// SIMATIC S7-200 project (STEP 7-Micro/WIN), CPU 226 REL 01.22

SYMBOL_TABLE USR1
Always_On        SM0.0    // This bit is always on.
First_Scan_On    SM0.1    // This bit is on for the first scan cycle only.
Clock_1s         SM0.5    // Clock pulse that is on for 0.5 s, off for 0.5 s, for a duty cycle time of 1 s.
Pot0_Value       SMB28    // Stores value entered by analog adjustment 0. Updated once per cycle in STOP/RUN
END_SYMBOL_TABLE

ORGANIZATION_BLOCK MAIN:OB1
TITLE=The system initializes on first startup, setting the TD 200 display state to 0 to show date and time, while initializing the pressure update speed to 50 (500ms), the pressure value to 12,345,678, and the output configuration to 0. Operators can use the TD 200 arrow keys to switch the display state, viewing different information such as date/time, pressure value, or motor status, with the state cycling between 0 and 6.
// When the display state is 1, operators can control pressure value updates via function keys F1-F4: F1 stops updates, F2 starts updates, F3 sets the update speed to 1 (10ms), and F4 sets it to 150 (1500ms). Pressure value updates are managed by a control flag and increment when the timer expires.
// If the display state is 2, F1 clears the output configuration to disable output points, F2 sets it to fully enabled, and F3 activates I/O cycling. The output configuration is set to fully enabled on the clock pulse rising edge and cleared on the falling edge.
// When the display state is 3, the system displays the analog potentiometer value in bar graph and numeric formats. For display state 4, the system supports scrolling message display, with F1-F4 setting the scroll speed to 1 (100ms), 5 (500ms), 10 (1000ms), or 15 (1500ms). In display state 6, it shows "ON 1" or "OFF 0" based on the motor status.
// The system supports a second TD 200 panel, with its display state controlling the content. State 0 shows the input byte in hexadecimal, decimal, and individual bit status, while state 1 shows the output byte’s equivalent information. 
BEGIN
Network 1 //  Initialize the Values to Be Used
//  Load SM0.1 to process this network in the first scan cycle only.
//  Move the hexadecimal value 8000 (binary 1000 0000 0000 0000) to variable
//  memory word VW12 to enable the first message on the TD 200 (device 1).
//  Move the constant 0 to variable memory word VW700 to set the
//  display state of the TD 200 to evaluate the function keys for
//  the pressure value (executed in subroutine SBR1).
//  Move the constant 0 to memory byte MB0 to clear the TD 200 function
//  key area.
//  Move the constant 0 to memory byte MB1 to clear the TD 200 help bit area.
//  Move the constant 50 to variable memory word VW704 to initialize
//  the embedded value for the pressure update speed.
//  Move the constant 12,345,678 to variable memory double word VD156
//  to set the pressure value.
//  Move the constant 0 to variable memory word VW706 to initialize
//  the output configuration with the function keys.
//  Fill the message area with full blocks in a bar graph.
//  Move 20 bytes starting from variable memory byte VB260 into VB900 to
//  copy the message to scroll on the TD 200 display.
//  Move the constant 15 to variable memory word VW800 to set the update
//  speed for the message scroll to slow.
//  Move the real number 1234.000 to variable memory double word VD316
//  to initialize the real value.
//  Move the hexadecimal value 80 (binary 1000 0000) to variable memory
//  byte VB512 to enable the second TD 200 (optional).
//  Move the constant 0 to variable memory word VW702 to set the
//  display state of the second TD 200 to zero.
// 
LD     First_Scan_On:SM0.1   // In the first scan cycle,
MOVW   16#8000, VW12         // enable the first message on
// device 1.
MOVW   +0, VW700             // Display the state of device 1
// set to zero.
MOVB   16#0, MB0             // Clear the function key area.
MOVB   16#0, MB1             // Clear the help bit area.
MOVW   +50, VW704            // Initialize the update speed (pressure)
MOVD   +12345678, VD156      // Set the pressure value.
MOVW   +0, VW706             // Initialize the I/O cycles.
FILL   16#FFFF, VW770, 10    // Fill the TD 200 message area
// with full blocks.
BMB    VB260, VB900, 20      // Copy the message to scroll.
MOVW   +15, VW800            // Set the scrolling update speed
// to slow.
MOVR   1234.0, VD316         // Initialize the real value.
MOVB   16#80, VB512          // Enable the first message on device
// 2.
MOVW   +0, VW702             // Set the display state of device
// 2 to zero.
Network 2 //  Set Up a Timer to Increment the Data Values
//  Load memory bit M1.0 to process this network (run the timer) only
//  when the pressure updates are running.
//  Start the retentive on-delay timer T1 with a preset time of the
//  value in variable memory word VW704. T1 has a resolution of 10 ms.
//  Each count of the current value is a multiple of that resolution.
//  For example, a count of 50 on a 10 ms timer represents 500 ms.
// 
LD     M1.0                  // Run timer only when the pressure
// updates are running.
TONR   T1, VW704             // Start timer T1 with a preset
// time of the value in VW704.
Network 3 //  Reset Timer T1 and Increment the Pressure Value
//  Load retentive on-delay timer T1 to process this network if the
//  timer has expired.
//  If the timer has expired,
//  reset the timer and
//  increment variable memory double word VD156 to increment the pressure
//  value.
// 
LD     T1                    // If timer T1 has expired,
R      T1, 1                 // reset the timer and
INCD   VD156                 // increment the pressure value.
Network 4 //  Subroutine SBR7
//  Special memory bit SM0.5 provides a clock pulse that is on for
//  0.5 s and off for 0.5 s, for a duty cycle time of 1 s.
//  Load SM0.5.
//  If there is a positive transition (Edge Up) at SM0.5,
//  move the hexadecimal value FFFF (binary 1111 1111 1111 1111) to variable
//  memory word VW706 to fill VW706 with ones and turn on the associated
//  outputs.
//  This subroutine writes a different text to the display, depending
//  on the status of input bit I0.0 (display state 6).
//  Start SBR6.
//  This subroutine reads the CPU input byte IB0 and displays
//  it in decimal format. The subroutine also displays the status of
//  each input bit (ON = 1, OFF = 0) on the TD 200 (device 2 display
//  state 0).
//  Start SBR7.
// 
LD     Clock_1s:SM0.5        // If the 0.5 s clock pulse value
EU                           // changes from 0 to 1,
MOVW   16#FFFF, VW706        // fill VW706 with ones to cycle
// on the outputs.
Network 5 //  Subroutine SBR4
//  Load SM0.5.
//  If there is a negative transition (Edge Down) at SM0.5,
//  move the hexadecimal value 0 to variable memory word VW706 to fill
//  VW706 with zeros and turn off the associated outputs.
//  This subroutine handles the memory bits set by the
//  TD 200 function keys (display state 1).
//  Start SBR1.
//  This subroutine writes a text message on the first row of the
//  TD 200 display and scrolls it to the left at the speed selected
//  (display state 4).
//  Start SBR4.
// 
LD     Clock_1s:SM0.5        // If the 0.5 s clock pulse value
ED                           // changes from 1 to 0,
MOVW   16#0, VW706           // fill VW706 with zeros to cycle
// off the outputs.
Network 6 //  Write the Values in Variable Memory Word VW706 to Outputs
//  Load memory bit M1.2 to process this network if the I/O cycle
//  process is enabled.
//  Move the value in VW706 to output word QW0.
// 
LD     M1.2                  // If the I/O cycles are enabled,
MOVW   VW706, QW0            // write to the outputs.
Network 7 //  If the TD 200 Display State Is 0, Call Subroutine SBR0
//  If the value in variable memory word VW700 is 0 (TD 200 menu 1 selected),
//  call subroutine SBR0 to display the date and time.
// 
LDW=   VW700, +0             // If the TD 200 display state = 0,
CALL   SBR_0:SBR0            // call SBR0.
Network 8 //  Subroutine SBR3
//  Check the value in memory byte MB0 to see if a function key on the
//  TD 200 has been pressed.
//  If the value in memory byte MB0 is not equal to 0
//  and the value in variable memory word VW700 is 1 (TD 200 menu 2 selected),
//  call subroutine SBR1 to evaluate the function keys to change
//  the pressure value.
//  This subroutine handles the function keys for the output configuration
//  (display state 2).
//  Start SBR2.
//  This subroutine contains the logic to display the analog adjustment
//  (POT) 0 in the form of a bar chart (display state 3). You can use
//  a small screwdriver to change the value of the POT.
//  Start SBR3.
// 
LDB=   MB0, 0                // If a function key
NOT                          // is pressed (MB0 not equal 0)
AW=    VW700, +1             // and the TD 200 display state  = 1,
CALL   SBR_1:SBR1            // call SBR1.
Network 9 //  If the TD 200 Display State Is 2, Call Subroutine SBR2
//  Check the value in memory byte MB0 to see if a function key on the
//  TD 200 has been pressed.
//  If the value in memory byte MB0 is not equal to 0
//  and the value in variable memory word VW700 is 2 (TD 200 menu 3 selected),
//  call subroutine SBR2 to evaluate the function keys to for the
//  output configuration.
// 
LDB=   MB0, 0                // If a function key
NOT                          // is pressed (MB0 not equal 0)
AW=    VW700, +2             // and the TD 200 display state = 2,
CALL   SBR_2:SBR2            // call SBR2.
Network 10 //  Subroutine SBR5
//  If the value in variable memory word VW700 is 3 (TD 200 menu 4 selected),
//  call subroutine SBR3 to update the analog adjustment (POT) value
//  as a bar chart graphic and in decimal form.
//  This subroutine clears the memory bits associated with the
//  TD 200 function keys. This allows a TD 200 system routine to edit
//  a real value after the ENTER key is pressed (display state 5).
//  Start SBR5.
// 
LDW=   VW700, +3             // If the TD 200 display state = 3,
CALL   SBR_3:SBR3            // call SBR3.
Network 11 //  If the TD 200 Display State Is 4, Call Subroutine SBR4
//  If the value in variable memory word VW700 is 4 (TD 200 menu 5 selected),
//  call subroutine SBR4 to scroll and display a message on the TD 200.
// 
LDW=   VW700, +4             // If the TD 200 display state = 4,
CALL   SBR_4:SBR4            // call SBR4.
Network 12 //  If the TD 200 Display State Is 5, Call Subroutine SBR5
//  If the value in variable memory word VW700 is 5 (TD 200 menu 6 selected),
//  call subroutine SBR5 to clear the memory bits of the function
//  keys.
// 
LDW=   VW700, +5             // If the TD 200 display state = 5,
CALL   SBR_5:SBR5            // call SBR5.
Network 13 //  Subroutine SBR8
//  If the value in variable memory word VW700 is 6 (TD 200 menu 7 selected),
//  call subroutine SBR6 to display the state of the motor (ON/OFF) on
//  the TD 200.
//  This subroutine reads the CPU output byte QB0 and displays
//  it in decimal format. The subroutine also displays the status of
//  each output bit (ON = 1, OFF = 0) on the TD 200 (device 2 display
//  state 1).
//  Start SBR8.
// 
LDW=   VW700, +6             // If the TD 200 display state = 6,
CALL   SBR_6:SBR6            // call SBR6.
Network 14 //  If the Second TD 200 Display State Is 0, Call Subroutine SBR7
//  If the value in variable memory word VW702 is 0 (second TD 200 menu
//  1 selected),
//  call subroutine SBR7 to update and display the CPU inputs.
// 
LDW=   VW702, +0             // If the second TD 200 display
// state = 0,
CALL   SBR_7:SBR7            // call SBR7.
Network 15 //  If the Second TD 200 Display State Is 1, Call Subroutine SBR8
//  If the value in variable memory word VW702 is 1 (second TD 200
//  menu 2 selected),
//  call subroutine SBR8 to update and display the CPU outputs.
// 
LDW=   VW702, +1             // If the second TD 200 display
// state = 1,
CALL   SBR_8:SBR8            // call SBR8.
Network 16 //  If the UP ARROW Is Pressed, Increment the Display State
//  Evaluate the arrow keys of the TD 200 device 1.
//  The first parameter block begins at VW0. The arrow keys are associated
//  with the fourth byte of the parameter block.
//  Load variable memory bit V3.3 to evaluate the UP ARROW key of the
//  TD 200.
//  If the UP ARROW key is pressed,
//  reset variable memory bit V3.3 and
//  increment variable memory word VW700 to change to the next TD 200
//  display state (move to the next TD 200 menu)
// 
LD     V3.3                  // If the UP ARROW key is pressed,
R      V3.3, 1               // reset V3.3 and
INCW   VW700                 // increment VW700.
Network 17 //  If the TD 200 Display State Moves above 6, Reset to 0
//  If the display state of the TD 200 = 7,
//  move the constant 0 to variable memory bit VW700 to change the
//  display state to 0.
// 
LDW=   VW700, +7             // If VW700 = 7,
MOVW   +0, VW700             // set the TD 200 display state = 0.
Network 18 //  If the DOWN ARROW Is Pressed, Decrement the Display State
//  Evaluate the arrow keys of the TD 200 device 1.
//  The first parameter block begins at VW0, The arrow keys are associated
//  with the fourth byte of the parameter block.
//  Load variable memory bit V3.2 to evaluate the DOWN ARROW key of the
//  TD 200.
//  If the DOWN ARROW key is pressed,
//  reset variable memory bit V3.2 and
//  decrement variable memory word VW700 to change to the previous TD 200
//  display state (move to the previous TD 200 menu)
// 
LD     V3.2                  // If the DOWN ARROW key is pressed,
R      V3.2, 1               // reset V3.2 and
DECW   VW700                 // decrement VW700.
Network 19 //  If the TD 200 Display State Moves below 0, Reset to 6
//  If the display state of the TD 200 = -1,
//  move the constant 6 to VW700 to change the display state to 6.
// 
LDW<=  VW700, -1             // If VW700 = -1,
MOVW   +6, VW700             // set the TD 200 display state = 6.
Network 20 //  If the UP ARROW Is Pressed, Increment the Display State of the Second Device
//  Evaluate the arrow keys of the TD 200 device 2.
//  The second device parameter block begins at VW500, The arrow
//  keys are associated with the fourth byte of the parameter block.
//  Load variable memory bit V503.3 to evaluate the UP ARROW key of the
//  second TD 200.
//  If the UP ARROW key is pressed,
//  reset variable memory bit V503.3 and
//  increment variable memory word VW702 to change to the next TD 200
//  display state (move to the next TD 200 menu)
// 
LD     V503.3                // If the UP ARROW key is pressed,
R      V503.3, 1             // reset V503.3 and
INCW   VW702                 // increment VW702.
Network 21 //  If the Second TD 200 Display State Moves above 1, Reset to 0
//  If the display state of the second TD 200 = 2,
//  move the constant 0 to variable memory bit VW702 to change the
//  display state to 0.
// 
LDW=   VW702, +2             // If VW702 = 2,
MOVW   +0, VW702             // set the TD 200 display state = 0.
Network 22 //  If the DOWN ARROW Is Pressed, Decrement the Display State of the Second Device
//  Evaluate the arrow keys of the TD 200 device 2.
//  The first parameter block begins at VW500, The arrow keys are associated
//  with the fourth byte of the parameter block.
//  Load variable memory bit V503.2 to evaluate the DOWN ARROW key of the
//  TD 200.
//  If the DOWN ARROW key is pressed,
//  reset variable memory bit V503.2 and
//  decrement variable memory word VW702 to change to the previous TD 200
//  display state (move to the previous TD 200 menu).
// 
LD     V503.2                // If the DOWN ARROW key is pressed,
R      V503.2, 1             // reset V503.2 and
DECW   VW702                 // decrement VW702.
Network 23 //  If the TD 200 Display State Moves below 0, Reset to 1
//  If the display state of the second TD 200 = -1,
//  move the constant 1 to VW702 to change the display state to 1.
// 
LDW<=  VW702, -1             // If VW702 = -1,
MOVW   +1, VW702             // set the TD 200 diplay state = 1.
Network 24 //  Set the Message Enable Bit Based on the Current Display State
//  Load special memory bit SM0.0 to process this network every scan cycle.
//  Move the hexadecimal value 8000 (binary 1000 0000 0000 0000) to
//  variable memory word VW12 to set the first message enable bit (V12.7)
//  Shift the value in VW12 by the value in variable memory byte VB701
//  (least significant byte of the display state variable memory word).
//  This sets the message enable bit that corresponds to the display state.
// 
LD     Always_On:SM0.0       // Every scan cycle,
MOVW   16#8000, VW12         // enable the first message
// on device 1.
SRW    VW12, VB701           // Shift the value in VW12 based on
// the value in VB701.
Network 25 //  Set the Message Enable Bit Based on the Current Display State of Device 2
//  Load special memory bit SM0.0 to process this network every scan cycle
//  Move the hexadecimal value 8000 (binary 1000 0000 0000 0000) to
//  variable memory word VW512 to set the first message enable bit (V512.7)
//  for the second TD 200 device.
//  Shift the value in VW512 by the value in variable memory byte VB703
//  (lest significant byte of the display state variable memory word).
//  This sets the message enable bit that corresponds to the display state
//  of the second device.
// 
LD     Always_On:SM0.0       // Every scan cycle,
MOVW   16#8000, VW512        // enable the first message
// on device 2.
SRW    VW512, VB703          // Shift the value in VW512 based on
// the value in VB703.
Network 26 //  Main Program End
//  End the main program.
// MEND					// End the main program.
// 
// ***SUBROUTINES***
// 
// 
Network 27 //  Subroutine SBR0
//  Start SBR0 to display the date and time on the TD 200 device 1.
// 
END_ORGANIZATION_BLOCK

SUBROUTINE_BLOCK SBR_0:SBR0
TITLE=
BEGIN
Network 2 //  Get and Display the Date
//  Load special memory bit SM0.0 to process this network every scan cycle.
//  Read the current time and date and load it in variable memory
//  byte VB720.
//  Starting at variable memory byte VB721, convert two hexadecimal digits
//  to an ASCII string and store the result at variable memory byte
//  VB100. This converts the month for display on the TD 200.
//  Move the hexadecimal value 2D to variable memory byte VB102 to
//  load a "-" to the TD 200 display.
//  Starting at variable memory byte VB722, convert two hexadecimal digits
//  to an ASCII string and store the result at variable memory byte
//  VB103. This converts the day of the month for display on the TD 200.
//  Move the hexadecimal value 2D to variable memory byte VB105 to
//  load a "-" to the TD 200 display.
//  Starting at variable memory byte VB720, convert two hexadecimal digits
//  to an ASCII string and store the result at variable memory byte
//  VB106. This converts the year for display on the TD 200.
//  Move the hexadecimal value 2020 to variable memory word VW108 to
//  load two blank spaces to the TD 200 display.
//  Move the hexadecimal value 2020 to variable memory word VW110 to
//  load two more blank spaces to the TD 200 display.
// 
LD     Always_On:SM0.0       // Every scan cycle,
TODR   VB720                 // read the real-time clock.
HTA    VB721, VB100, 2       // Convert the month to ASCII
// and display on the TD 200.
MOVB   16#2D, VB102          // Load a "-" for display.
HTA    VB722, VB103, 2       // Convert the day of the month
// and display.
MOVB   16#2D, VB105          // Load a "-" for display.
HTA    VB720, VB106, 2       // Convert the year to ASCII
// and display.
MOVW   16#2020, VW108        // Load two blanks.
MOVW   16#2020, VW110        // Load two blanks.
Network 3 //  Get and Display the Time
//  Load special memory bit SM0.0 to process this network every scan cycle.
//  Starting at variable memory byte VB723, convert two hexadecimal digits
//  to an ASCII string and store the result at variable memory byte
//  VB112. This converts the hour for display on the TD 200.
//  Move the hexadecimal value 3A to variable memory byte VB114 to
//  load a ":" to the TD 200 display.
//  Starting at variable memory byte VB724, convert two hexadecimal digits
//  to an ASCII string and store the result at variable memory byte
//  VB115. This converts the minutes for display on the TD 200.
//  Move the hexadecimal value 3A to variable memory byte VB117 to
//  load a ":" to the TD 200 display.
//  Starting at variable memory byte VB725, convert two hexadecimal digits
//  to an ASCII string and store the result at variable memory byte
//  VB118. This converts the seconds for display on the TD 200.
// 
LD     Always_On:SM0.0       // Every scan cycle,
HTA    VB723, VB112, 2       // convert the hour to ASCII
// and display on the TD 200.
MOVB   16#3A, VB114          // Load a ":" for display.
HTA    VB724, VB115, 2       // Convert the minutes to ASCII
// and display on the TD 200.
MOVB   16#3A, VB117          // Load a ":" for display.
HTA    VB725, VB118, 2       // Convert the seconds to ASCII
// and display on the TD 200.
Network 4 //  End of Subroutine SBR0
//  End SBR0.
// RET					// End SBR0.
// 
END_SUBROUTINE_BLOCK

SUBROUTINE_BLOCK SBR_1:SBR1
TITLE=
BEGIN
Network 2 //  Press F1 to Stop the Pressure Updates
//  Load memory bit M0.0 to check the status of the TD 200 function
//  key F1.
//  If memory bit M0.0 is set (F1 function key was pressed),
//  reset memory bit M1.0 to stop the pressure updates.
// 
LD     M0.0                  // If the F1 key has been pressed,
R      M1.0, 1               // stop the pressure updates.
Network 3 //  Press F2 to Start the Pressure Updates
//  Load memory bit M0.1 to check the status of the TD 200 function
//  key F2.
//  If memory bit M0.1 is set (F2 function key was pressed),
//  set memory bit M1.0 to start the pressure updates.
// 
LD     M0.1                  // If the F2 key has been pressed,
S      M1.0, 1               // start the pressure updates.
Network 4 //  Press F3 to Set the Pressure Readings for Fast Updates
//  Load memory bit M0.2 to check the status of the TD 200 function
//  key F3.
//  If memory bit M0.2 is set (F3 function key was pressed),
//  move the constant 1 to variable memory word VW704 to set the pressure
//  update speed to fast.
//  The value in VW704 is used as the preset time in the retentive
//  on-delay timer T1 (see Network 2). T1 has a resolution of 10 ms.
//  This means that a preset time (PT) of 1 results in a 10-ms timer.
// 
LD     M0.2                  // If the F3 key has been pressed,
MOVW   +1, VW704             // set the pressure readings for
// fast updates (10 ms).
Network 5 //  Press F4 to Set the Pressure Readings for Slow Updates
//  Load memory bit M0.3 to check the status of the TD 200 function
//  key F4.
//  If memory bit M0.3 is set (F4 function key was pressed),
//  move the constant 150 to variable memory word VW704 to set the pressure
//  update speed to slow.
//  The value in VW704 is used as the preset time in the retentive
//  on-delay timer T1 (see Network 2). T1 has a resolution of 10 ms.
//  This means that a preset time (PT) of 150 results in a 1500-ms
//  timer.
// 
LD     M0.3                  // If the F4 key has been pressed,
MOVW   +150, VW704           // set the pressure readings for
// slow updates (1500 ms).
Network 6 //  Clear the Function Key Area
//  Load special memory bit SM0.0 to process this network every scan cycle.
//  Move the constant 0 to memory byte MB0 to clear the function key
//  area.
// 
LD     Always_On:SM0.0       // Every scan cycle,
MOVB   0, MB0                // clear the function key area.
Network 7 //  End of Subroutine SBR1
//  End SBR1.
// RET					// End SBR1.
// 
END_SUBROUTINE_BLOCK

SUBROUTINE_BLOCK SBR_2:SBR2
TITLE=
BEGIN
Network 2 //  Stop the I/O Cycles
//  Load special memory bit SM0.0 to process this network every scan cycle.
//  Reset memory bit M1.2 to stop the I/O cycles.
// 
LD     Always_On:SM0.0       // Every scan cycle,
R      M1.2, 1               // stop the I/0 cycles.
Network 3 //  Press F1 to Disable All Outputs
//  Load memory bit M0.0 to check the status of the TD 200 function
//  key F1.
//  If memory bit M0.0 is set (F1 function key was pressed),
//  move the constant 0 to output word QW0 to disable the output
//  bits Q0.0 to Q0.7.
// 
LD     M0.0                  // If the F1 key has been pressed,
MOVW   +0, QW0               // disable all the outputs.
Network 4 //  Press F2 to Set All Outputs
//  Load memory bit M0.1 to check the status of the TD 200 function
//  key F2.
//  If memory bit M0.1 is set (F2 function key was pressed),
//  move the hexadecimal value FFFF (binary 1111 1111 1111 1111) to
//  output word QW0 to set the output bits Q0.0 to Q0.7.
// 
LD     M0.1                  // If the F2 key has been pressed,
MOVW   16#FFFF, QW0          // set all the outputs.
Network 5 //  Press F3 to Enable I/O Cycles
//  Load memory bit M0.2 to check the status of the TD 200 function
//  key F3.
//  If memory bit M0.2 is set (F3 function key was pressed),
//  set memory bit M1.2 to enable the I/O cycles.
// 
LD     M0.2                  // If the F3 key has been pressed,
S      M1.2, 1               // enable I/O cycles.
Network 6 //  Clear the Function Key Area
//  Load special memory bit SM0.0 to process this network every scan cycle.
//  Move the constant 0 to memory byte MB0 to clear the function key
//  area.
// 
LD     Always_On:SM0.0       // Every scan cycle,
MOVB   0, MB0                // clear the function key area.
Network 7 //  End of Subroutine SBR2
//  End SBR2.
// RET					// End SBR2.
// 
END_SUBROUTINE_BLOCK

SUBROUTINE_BLOCK SBR_3:SBR3
TITLE=
BEGIN
Network 2 //  Display the POT Value as a Bar Chart
//  Load special memory bit SM0.0 to process this network every scan cycle.
//  Starting at variable memory word VW240, fill the next 10 words with
//  the hexadecimal value 2020 to fill the message space with blanks.
//  Move the constant 0 to variable memory double word VD750 to clear
//  a space for the following calculations.
//  Special memory byte SMB28 stores the value entered with analog
//  adjustment 0 (POT 0). This value is updated once per scan cycle
//  in STOP/RUN.
//  Move the POT value from SMB28 to VB753.
//  Move the POT value from VB753 to VB239 to display the POT value
//  on the first row of the TD 200 display.
//  Divide the value in VD752 by 13 (20 characters * 13 > 256) and
//  place the remainder in VD750.
//  Move the remainder from VD750 to VW762.
//  Move the constant 0 to VW760 to clear the most significant byte.
//  Divide the remainder in VW762 by 3 to get a reading of fifths.
//  Starting at VB770, move the number of bytes specified in VB753
//  to VB240 for display.
//  Set variable memory double word VD770 to function as a pointer
//  to variable memory byte VB240 by moving &VB240 into VD790.
//  (The & in front of VB240 indicates that you are moving the address of
//  this memory location to VD790. VD790 then acts as a pointer to
//  this location.)
//  Add the value in VW752 to VW792 to offset to the first space.
//  Add the hexadecimal value FA (binary 1111 1010) to the value
//  in VW762 to create a character.
//  Move the value in VB763 to the location pointed to by variable
//  memory double word VD790. (The asterisk in front of VD790 indicates
//  that the contents of this double word are a pointer to another
//  location in memory, namely the TD 200 display buffer).
// 
LD     Always_On:SM0.0       // Every scan cycle,
FILL   16#2020, VW240, 10    // fill the message space with blanks.
MOVD   +0, VD750             // Clear a space to work in variable
// memory.
MOVB   Pot0_Value:SMB28, VB753 // Get the value of POT 0.
MOVB   VB753, VB239          // Display the POT value on the
// first row of the TD 200 display.
DIV    +13, VD750            // Divide the POT value by 13
// (20 character * 13 > 256).
MOVW   VW750, VW762          // Get the remainder.
MOVW   +0, VW760             // Clear the most significant byte.
DIV    +3, VD760             // Divide the remainder by 3 to
// get fifths.
BMB    VB770, VB240, VB753   // Move the full bars to the display
// buffer.
MOVD   &VB240, VD790         // Create a pointer to the start
// of the display buffer.
+I     VW752, VW792          // Offset to the first space.
+I     16#FA, VW762          // Create a character.
MOVB   VB763, *VD790         // Store the partial block to
// the display buffer.
Network 3 //  Clear the Function Key Area
//  Load special memory bit SM0.0 to process this network every scan cycle.
//  Move the constant 0 to memory byte MB0 to clear the function key
//  area.
// 
LD     Always_On:SM0.0       // Every scan cycle,
MOVB   0, MB0                // clear the function key area.
Network 4 //  End of Subroutine SBR3
//  End SBR3.
// RET					// End SBR3.
// 
END_SUBROUTINE_BLOCK

SUBROUTINE_BLOCK SBR_4:SBR4
TITLE=
BEGIN
Network 2 //  Copy the Message Text to the Work Area and Start Timer
//  Load special memory bit SM0.0 to process this network every scan cycle.
//  Starting at variable memory byte VB260, move 20 bytes to the
//  variable memory area starting at VB900.
//  Start the retentive on-delay timer T31 with the preset value stored
//  in variable memory word VW800. T31 has a resolution of 100 ms.
//  Each count of the current value is a multiple of that resolution.
//  For example, a count of 5 on a 100 ms timer represents 500 ms.
// 
LD     Always_On:SM0.0       // Every scan cycle,
BMB    VB260, VB900, 20      // copy the text of the message
// to the work area.
TONR   T31, VW800            // Start timer T31 with a preset
// time (PT) of the value in
// VW800.
Network 3 //  After Timer Expires, Display Message and Begin Scrolling
//  Load retentive on-delay timer T31 to process this network if the
//  timer has expired.
//  If T31 has expired,
//  reset the timer.
//  Starting at variable memory byte VB901, move 19 bytes to variable
//  memory byte 260 to display characters 2 through 20 of the message
//  text.
//  Starting at variable memory byte VB900, move 1 byte to variable
//  memory byte 260 to display the first character of the message at
//  the end of the display line.
// 
LD     T31                   // If the timer has expired,
R      T31, 1                // reset the timer.
BMB    VB901, VB260, 19      // Display the last 19 characters
// of the message text.
BMB    VB900, VB279, 1       // Display the first character
// of the text at the end of the
// message.
Network 4 //  Press F1 for Fastest Scroll
//  Load memory bit M0.0 to check the status of the TD 200 function
//  key F1.
//  If memory bit M0.0 is set (F1 function key was pressed),
//  move the constant 1 to variable memory word VW800 to set the
//  message scrolling speed to fastest.
//  The value in VW800 is used as the preset time in the retentive
//  on-delay timer T31 (see Network 50). T31 has a resolution of 100 ms.
//  This means that a preset time (PT) of 1 results in a 100-ms timer.
// 
LD     M0.0                  // If the F1 key has been pressed,
MOVW   +1, VW800             // set the scrolling to fastest.
Network 5 //  Press F2 for Fast Scroll
//  Load memory bit M0.1 to check the status of the TD 200 function
//  key F2.
//  If memory bit M0.1 is set (F2 function key was pressed),
//  move the constant 5 to variable memory word VW800 to set the
//  message scrolling speed to fast.
//  The value in VW800 is used as the preset time in the retentive
//  on-delay timer T31 (see Network 50). T31 has a resolution of 100 ms.
//  This means that a preset time (PT) of 5 results in a 500-ms timer.
// 
LD     M0.1                  // If the F2 key has been pressed,
MOVW   +5, VW800             // set the scrolling to fast.
Network 6 //  Press F3 for Slow Scroll
//  Load memory bit M0.2 to check the status of the TD 200 function
//  key F3.
//  If memory bit M0.2 is set (F3 function key was pressed),
//  move the constant 10 to variable memory word VW800 to set the
//  message scrolling speed to slow.
//  The value in VW800 is used as the preset time in the retentive
//  on-delay timer T31 (see Network 50). T31 has a resolution of 100 ms.
//  This means that a preset time (PT) of 10 results in a 1000-ms timer.
// 
LD     M0.2                  // If the F3 key has been pressed,
MOVW   +10, VW800            // set the scrolling to slow.
Network 7 //  Press F3 for Slowest Scroll
//  Load memory bit M0.3 to check the status of the TD 200 function
//  key F4.
//  If memory bit M0.3 is set (F4 function key was pressed),
//  move the constant 15 to variable memory word VW800 to set the
//  message scrolling speed to slowest.
//  The value in VW800 is used as the preset time in the retentive
//  on-delay timer T31 (see Network 50). T31 has a resolution of 100 ms.
//  This means that a preset time (PT) of 15 results in a 1500-ms timer.
// 
LD     M0.3                  // If the F4 key has been pressed,
MOVW   +15, VW800            // set the scrolling to slowest.
Network 8 //  Clear the Function Key Area
//  Load special memory bit SM0.0 to process this network every scan cycle.
//  Move the constant 0 to memory byte MB0 to clear the function key
//  area.
// 
LD     Always_On:SM0.0       // Every scan cycle,
MOVB   0, MB0                // clear the function key area.
Network 9 //  End of Subroutine SBR4
//  End SBR4.
// RET					// End SBR4.
// 
END_SUBROUTINE_BLOCK

SUBROUTINE_BLOCK SBR_5:SBR5
TITLE=
BEGIN
Network 2 //  Clear the Function Key Area
//  Load special memory bit SM0.0 to process this network every scan cycle.
//  Move the constant 0 to memory byte MB0 to clear the function key
//  area.
// 
LD     Always_On:SM0.0       // Every scan cycle,
MOVB   0, MB0                // clear the function key area.
Network 3 //  End of Subroutine SBR5
//  End SBR5.
// RET					// End SBR5.
// 
END_SUBROUTINE_BLOCK

SUBROUTINE_BLOCK SBR_6:SBR6
TITLE=
BEGIN
Network 2 //  If Input Is On, Write "ON 1".  If Input Is Off, Write "OFF 0".
//  The message displayed on the TD 200 during display state 6 contains
//  an embedded message. The message is "MOTOR XXX  I0.0 = X." The logic
//  in this subroutine provides the appropriate characters for the
//  spaces marked with "X."
//  Load input I0.0.
//  If input I0.0 is on,
//  Move the hexadecimal value 4F to variable memory byte VB346 to display
//  the letter "O" in the first embedded text display area.
//  Move the hexadecimal value F3 to variable memory byte VB347 to display
//  the letter "N" in the second embedded text display area.
//  Move the hexadecimal value 20 to variable memory byte VB348 to display
//  a space in the third embedded text display area.
//  Move the hexadecimal value 31 to variable memory byte VB358 to display
//  a "1" in the final embedded text display area.
//  The complete message reads "Motor ON  I0.0 = 1."
//  If input I0.0 is not on,
//  Move the hexadecimal value 4F to variable memory byte 346 to display
//  the letter "O" in the first embedded text display area.
//  Move the hexadecimal value 46 to variable memory byte VB347 to display
//  the letter "F" in the second embedded text display area.
//  Move the hexadecimal value 46 to variable memory byte VB348 to display
//  the letter "F" in the third embedded text display area.
//  Move the hexadecimal value 30 to variable memory byte VB358 to display
//  a "0" in the final embedded text display area.
//  The complete message reads "Motor OFF I0.0 = 0."
// 
LD     I0.0                  // If input I0.0 is on,
MOVB   16#4F, VB346          // write 'O' to the display,
MOVB   16#4E, VB347          // write 'N' to the display,
MOVB   16#20, VB348          // write ' ' (space) to the display,
MOVB   16#31, VB358          // and write '1' to the display.
NOT                          // If input I0.0 is off,
MOVB   16#4F, VB346          // write 'O' to the display,
MOVB   16#46, VB347          // write 'F' to the display,
MOVB   16#46, VB348          // write 'F' to the display, and
MOVB   16#30, VB358          // write '0' to the display.
Network 3 //  End of Subroutine SBR6
//  End SBR6.
// RET					// End SBR6.
// 
END_SUBROUTINE_BLOCK

SUBROUTINE_BLOCK SBR_7:SBR7
TITLE=
BEGIN
Network 2 //  Convert Input Byte From Hexadecimal and Display
//  Load special memory bit SM0.0 to process this network every scan cycle.
//  Convert input byte IB0 from hexadecimal to ASCII and store in
//  variable memory byte VB572.
//  Move the value in input byte IB0 to variable memory byte VB578 for
//  display on the TD 200.
// 
LD     Always_On:SM0.0       // Every scan cycle,
HTA    IB0, VB572, 2         // convert input byte IB0 from Hex
// to ASCII.
MOVB   IB0, VB578            // Display input byte IB0 in decimal
// format on the TD 200.
Network 3 //  Display Status of Input Bit I0.0
//  Load input bit I0.0.
//  If input bit I0.0 is on, move the hexadecimal value 31 to variable
//  memory byte VB562 to write a "1" to the appropriate location on
//  the TD 200 display.
//  If input bit I0.0 is off, move the hexadecimal value 30 to variable
//  memory byte VB562 to write a "0" to the appropriate location on
//  the TD 200 display.
// 
LD     I0.0                  // If I0.0 is on,
MOVB   16#31, VB562          // write "1" to the corresponding
// place on the TD 200 display.
NOT                          // If I0.0 is off,
MOVB   16#30, VB562          // write "0" to the corresponding
// place on the TD 200 display.
Network 4 //  Display Status of Input Bit I0.1
//  Load input bit I0.1.
//  If input bit I0.1 is on, move the hexadecimal value 31 to variable
//  memory byte VB563 to write a "1" to the appropriate location on
//  the TD 200 display.
//  If input bit I0.1 is off, move the hexadecimal value 30 to variable
//  memory byte VB563 to write a "0" to the appropriate location on
//  the TD 200 display.
// 
LD     I0.1                  // If I0.1 is on,
MOVB   16#31, VB563          // write "1" to the corresponding
// place on the TD 200 display.
NOT                          // If I0.1 is off,
MOVB   16#30, VB563          // write "0" to the corresponding
// place on the TD 200 display.
Network 5 //  Display Status of Input Bit I0.2
//  Load input bit I0.2.
//  If input bit I0.2 is on, move the hexadecimal value 31 to variable
//  memory byte VB564 to write a "1" to the appropriate location on
//  the TD 200 display.
//  If input bit I0.2 is off, move the hexadecimal value 30 to variable
//  memory byte VB564 to write a "0" to the appropriate location on
//  the TD 200 display.
// 
LD     I0.2                  // If I0.2 is on,
MOVB   16#31, VB564          // write "1" to the corresponding
// place on the TD 200 display.
NOT                          // If I0.2 is off,
MOVB   16#30, VB564          // write "0" to the corresponding
// place on the TD 200 display.
Network 6 //  Display Status of Input Bit I0.3
//  Load input bit I0.3.
//  If input bit I0.3 is on, move the hexadecimal value 31 to variable
//  memory byte VB565 to write a "1" to the appropriate location on
//  the TD 200 display.
//  If input bit I0.3 is off, move the hexadecimal value 30 to variable
//  memory byte VB565 to write a "0" to the appropriate location on
//  the TD 200 display.
// 
LD     I0.3                  // If I0.3 is on,
MOVB   16#31, VB565          // write "1" to the corresponding
// place on the TD 200 display.
NOT                          // If I0.3 is off,
MOVB   16#30, VB565          // write "0" to the corresponding
// place on the TD 200 display.
Network 7 //  Display Status of Input Bit I0.4
//  Load input bit I0.4.
//  If input bit I0.4 is on, move the hexadecimal value 31 to variable
//  memory byte VB566 to write a "1" to the appropriate location on
//  the TD 200 display.
//  If input bit I0.4 is off, move the hexadecimal value 30 to variable
//  memory byte VB566 to write a "0" to the appropriate location on
//  the TD 200 display.
// 
LD     I0.4                  // If I0.4 is on,
MOVB   16#31, VB566          // write "1" to the corresponding
// place on the TD 200 display.
NOT                          // If I0.4 is off,
MOVB   16#30, VB566          // write "0" to the corresponding
// place on the TD 200 display.
Network 8 //  Display Status of Input Bit I0.5
//  Load input bit I0.5.
//  If input bit I0.5 is on, move the hexadecimal value 31 to variable
//  memory byte VB567 to write a "1" to the appropriate location on
//  the TD 200 display.
//  If input bit I0.5 is off, move the hexadecimal value 30 to variable
//  memory byte VB567 to write a "0" to the appropriate location on
//  the TD 200 display.
// 
LD     I0.5                  // If I0.5 is on,
MOVB   16#31, VB567          // write "1" to the corresponding
// place on the TD 200 display.
NOT                          // If I0.5 is off,
MOVB   16#30, VB567          // write "0" to the corresponding
// place on the TD 200 display.
Network 9 //  Display Status of Input Bit I0.6
//  Load input bit I0.6.
//  If input bit I0.6 is on, move the hexadecimal value 31 to variable
//  memory byte VB568 to write a "1" to the appropriate location on
//  the TD 200 display.
//  If input bit I0.6 is off, move the hexadecimal value 30 to variable
//  memory byte VB568 to write a "0" to the appropriate location on
//  the TD 200 display.
// 
LD     I0.6                  // If I0.6 is on,
MOVB   16#31, VB568          // write "1" to the corresponding
// place on the TD 200 display.
NOT                          // If I0.6 is off,
MOVB   16#30, VB568          // write "0" to the corresponding
// place on the TD 200 display.
Network 10 //  Display Status of Input Bit I0.7
//  Load input bit I0.7.
//  If input bit I0.7 is on, move the hexadecimal value 31 to variable
//  memory byte VB569 to write a "1" to the appropriate location on
//  the TD 200 display.
//  If input bit I0.7 is off, move the hexadecimal value 30 to variable
//  memory byte VB569 to write a "0" to the appropriate location on
//  the TD 200 display.
// 
LD     I0.7                  // If I0.7 is on,
MOVB   16#31, VB569          // write "1" to the corresponding
// place on the TD 200 display.
NOT                          // If I0.7 is off,
MOVB   16#30, VB569          // write "0" to the corresponding
// place on the TD 200 display.
Network 11 //  Clear the Function Key Area
//  Load special memory bit SM0.0 to process this network every scan cycle.
//  Move the constant 0 to memory byte MB0 to clear the function key
//  area.
// 
LD     Always_On:SM0.0       // Every scan cycle,
MOVB   0, MB0                // clear the function key area.
Network 12 //  End of Subroutine SBR7
//  End SBR7.
// RET					// End SBR7.
// 
END_SUBROUTINE_BLOCK

SUBROUTINE_BLOCK SBR_8:SBR8
TITLE=
BEGIN
Network 2 //  Convert Output Byte from Hexadecimal and Display
//  Load special memory bit SM0.0 to process this network every scan cycle.
//  Convert output byte QB0 from hexadecimal to ASCII and store in
//  variable memory byte VB612.
//  Move the value in output byte QB0 to variable memory byte VB618 for
//  display on the TD 200.
// 
LD     Always_On:SM0.0       // Every scan cycle,
HTA    QB0, VB612, 2         // convert output byte QB0 from Hex
// to ASCII.
MOVB   QB0, VB618            // Display output byte QB0 in decimal
// format on the TD 200.
Network 3 //  Display Status of Output Bit Q0.0
//  Load output bit Q0.0.
//  If output bit Q0.0 is on, move the hexadecimal value 31 to variable
//  memory byte VB602 to write a "1" to the appropriate location on
//  the TD 200 display.
//  If output bit Q0.0 is off, move the hexadecimal value 30 to variable
//  memory byte VB602 to write a "0" to the appropriate location on
//  the TD 200 display.
// 
LD     Q0.0                  // If Q0.0 is on,
MOVB   16#31, VB602          // write "1" to the corresponding
// place on the TD 200 display.
NOT                          // If Q0.0 is off,
MOVB   16#30, VB602          // write "0" to the corresponding
// place on the TD 200 display.
Network 4 //  Display Status of Output Bit Q0.1
//  Load output bit Q0.1.
//  If output bit Q0.1 is on, move the hexadecimal value 31 to variable
//  memory byte VB603 to write a "1" to the appropriate location on
//  the TD 200 display.
//  If output bit Q0.1 is off, move the hexadecimal value 30 to variable
//  memory byte VB603 to write a "0" to the appropriate location on
//  the TD 200 display.
// 
LD     Q0.1                  // If Q0.1 is on,
MOVB   16#31, VB603          // write "1" to the corresponding
// place on the TD 200 display.
NOT                          // If Q0.1 is off,
MOVB   16#30, VB603          // write "0" to the corresponding
// place on the TD 200 display.
Network 5 //  Display Status of Output Bit Q0.2
//  Load output bit Q0.2.
//  If output bit Q0.2 is on, move the hexadecimal value 31 to variable
//  memory byte VB604 to write a "1" to the appropriate location on
//  the TD 200 display.
//  If output bit Q0.2 is off, move the hexadecimal value 30 to variable
//  memory byte VB604 to write a "0" to the appropriate location on
//  the TD 200 display.
// 
LD     Q0.2                  // If Q0.2 is on,
MOVB   16#31, VB604          // write "1" to the corresponding
// place on the TD 200 display.
NOT                          // If Q0.2 is off,
MOVB   16#30, VB604          // write "0" to the corresponding
// place on the TD 200 display.
Network 6 //  Display Status of Output Bit Q0.3
//  Load output bit Q0.3.
//  If output bit Q0.3 is on, move the hexadecimal value 31 to variable
//  memory byte VB605 to write a "1" to the appropriate location on
//  the TD 200 display.
//  If output bit Q0.3 is off, move the hexadecimal value 30 to variable
//  memory byte VB605 to write a "0" to the appropriate location on
//  the TD 200 display.
// 
LD     Q0.3                  // If Q0.3 is on,
MOVB   16#31, VB605          // write "1" to the corresponding
// place on the TD 200 display.
NOT                          // If Q0.3 is off,
MOVB   16#30, VB605          // write "0" to the corresponding
// place on the TD 200 display.
Network 7 //  Display Status of Output Bit Q0.4
//  Load output bit Q0.4.
//  If output bit Q0.4 is on, move the hexadecimal value 31 to variable
//  memory byte VB606 to write a "1" to the appropriate location on
//  the TD 200 display.
//  If output bit Q0.4 is off, move the hexadecimal value 30 to variable
//  memory byte VB606 to write a "0" to the appropriate location on
//  the TD 200 display.
// 
LD     Q0.4                  // If Q0.4 is on,
MOVB   16#31, VB606          // write "1" to the corresponding
// place on the TD 200 display.
NOT                          // If Q0.4 is off,
MOVB   16#30, VB606          // write "0" to the corresponding
// place on the TD 200 display.
Network 8 //  Display Status of Output Bit Q0.5
//  Load output bit Q0.5.
//  If output bit Q0.5 is on, move the hexadecimal value 31 to variable
//  memory byte VB607 to write a "1" to the appropriate location on
//  the TD 200 display.
//  If output bit Q0.5 is off, move the hexadecimal value 30 to variable
//  memory byte VB607 to write a "0" to the appropriate location on
//  the TD 200 display.
// 
LD     Q0.5                  // If Q0.5 is on,
MOVB   16#31, VB607          // write "1" to the corresponding
// place on the TD 200 display.
NOT                          // If Q0.5 is off,
MOVB   16#30, VB607          // write "0" to the corresponding
// place on the TD 200 display.
Network 9 //  Display Status of Output Bit Q0.6
//  Load output bit Q0.6.
//  If output bit Q0.6 is on, move the hexadecimal value 31 to variable
//  memory byte VB608 to write a "1" to the appropriate location on
//  the TD 200 display.
//  If output bit Q0.6 is off, move the hexadecimal value 30 to variable
//  memory byte VB608 to write a "0" to the appropriate location on
//  the TD 200 display.
// 
LD     Q0.6                  // If Q0.6 is on,
MOVB   16#31, VB608          // write "1" to the corresponding
// place on the TD 200 display.
NOT                          // If Q0.6 is off,
MOVB   16#30, VB608          // write "0" to the corresponding
// place on the TD 200 display.
Network 10 //  Display Status of Output Bit Q0.7
//  Load output bit Q0.7.
//  If output bit Q0.7 is on, move the hexadecimal value 31 to variable
//  memory byte VB609 to write a "1" to the appropriate location on
//  the TD 200 display.
//  If output bit Q0.7 is off, move the hexadecimal value 30 to variable
//  memory byte VB609 to write a "0" to the appropriate location on
//  the TD 200 display.
// 
LD     Q0.7                  // If Q0.7 is on,
MOVB   16#31, VB609          // write "1" to the corresponding
// place on the TD 200 display.
NOT                          // If Q0.7 is off,
MOVB   16#30, VB609          // write "0" to the corresponding
// place on the TD 200 display.
Network 11 //  Clear the Function Key Area
//  Load special memory bit SM0.0 to process this network every scan cycle.
//  Move the constant 0 to memory byte MB0 to clear the function key
//  area.
// 
LD     Always_On:SM0.0       // Every scan cycle,
MOVB   0, MB0                // clear the function key area.
Network 12 //  End of Subroutine SBR8
//  End SBR8.
// RET					// End SBR8.
// 
END_SUBROUTINE_BLOCK

DATA_BLOCK_TAB USER1
BEGIN
//Data Block DB1 (V Memory):
// BEGIN TD200_BLOCK 0
// (Comments within this block should not be edited or removed)
VB0      'TD'                // TD 200 Identification
VB2      16#90               // Set Language to English, set Update to As fast as possible
VB3      16#71               // Set the display to 40 character mode; Up key V3.3; Down key V3.2
VB4      7                   // Set the number of messages
VB5      0                   // Set the Function Keys notification bits to M0.0 - M0.7 
VW6      100                 // Set the starting address for messages to VW100
VW8      12                  // Set the starting address for message enable bits to VW12
VW10     1000                // Global Password
// MESSAGE 1
// Message Enable Bit V12.7
VB100    '                    ARROW KEYS TO SCROLL'
// MESSAGE 2
// Message Enable Bit V12.6
VB140    'PRESSURE =    '
VB154    16#0                // No Edit; No Acknowledgement; No Password;
VB155    16#43               // Unsigned Double Word;  3 Digits to the right of the decimal;
VD156    16#0                // Embedded Data Value: Move data for display here.
VB160    'STOP  RUN  FAST SLOW'
// MESSAGE 3
// Message Enable Bit V12.5
VB180    'OUTPUT CONFIGURATIONOFF   ON   CYCL     '
// MESSAGE 4
// Message Enable Bit V12.4
VB220    '0   POT VALUE   '
VB236    16#0                // No Edit; No Acknowledgement; No Password;
VB237    16#30               // Unsigned Word;  0 Digits to the right of the decimal;
VW238    16#0                // Embedded Data Value: Move data for display here.
VB240    '                    '
// MESSAGE 5
// Message Enable Bit V12.3
VB260    '  This is a test!   FAST  FA-  SL+  SLOW'
// MESSAGE 6
// Message Enable Bit V12.2
VB300    'REAL VALUE:   '
VB314    16#18               // Edit Notification V314.2; No Acknowledgement;
// Edit Requires Password;
VB315    16#53               // Real Double Word;  3 Digits to the right of the decimal;
VD316    16#0                // Embedded Data Value: Move data for display here.
VB320    'Press ENTER to EDIT '
// MESSAGE 7
// Message Enable Bit V12.1
VB340    'Motor      I0.0 =   Use I0.0 to toggle  '
// END TD200_BLOCK 0
// BEGIN TD200_BLOCK 500
// (Comments within this block should not be edited or removed)
VB500    'TD'                // TD 200 Identification
VB502    16#90               // Set Language to English, set Update to As fast as possible
VB503    16#71               // Set the display to 40 character mode; Up key V503.3; 
// Down key V503.2
VB504    2                   // Set the number of messages
VB505    0                   // Set the Function Keys notification bits to M0.0 - M0.7 
VW506    540                 // Set the starting address for messages to VW540
VW508    512                 // Set the starting address for message enable bits to VW512
VW510    1000                // Global Password
// MESSAGE 1
// Message Enable Bit V512.7
VB540    'Display Inputs      I:XXXXXXXXb XXh'
VB575    16#0                // No Edit; No Acknowledgement; No Password;
VB576    16#30               // Unsigned Word;  0 Digits to the right of the decimal;
VW577    16#0                // Embedded Data Value: Move data for display here.
VB579    'd'
// MESSAGE 2
// Message Enable Bit V512.6
VB580    'Display Outputs     Q:XXXXXXXXb XXh'
VB615    16#0                // No Edit; No Acknowledgement; No Password;
VB616    16#30               // Unsigned Word;  0 Digits to the right of the decimal;
VW617    16#0                // Embedded Data Value: Move data for display here.
VB619    'd'
// END TD200_BLOCK 500
END_DATA_BLOCK_TAB
